// TIA Portal project "TiaProject-SortColors" (V17)

(* hardware
DEVICE "S7-1200 station_1"  S7-1200 Station
   slot 0: "Rack_0"  S7-1200 Rack  Rack  V1.0
   slot 1: "Brain"  CPU 1212C AC/DC/Rly  6ES7 212-1BE40-0XB0  V4.5
*)

// ===== PLC "Brain"  CPU 1212C AC/DC/Rly =====

VAR_GLOBAL   // PLC tag table "Steps"
   "X0" AT %M1.0 : Bool;
   "X1" AT %M1.1 : Bool;
   "X2" AT %M1.2 : Bool;
   "X3" AT %M1.3 : Bool;
   "X4" AT %M1.4 : Bool;
   "X5" AT %M1.5 : Bool;
   "X6" AT %M1.6 : Bool;
   "X7" AT %M1.7 : Bool;
   "X8" AT %M6.0 : Bool;
   "X9" AT %M6.1 : Bool;
   "X10" AT %M6.2 : Bool;
   "X11" AT %M6.3 : Bool;
   "X12" AT %M6.4 : Bool;
END_VAR

VAR_GLOBAL   // PLC tag table "I/O"
   "i1" AT %I0.0 : Bool;   // Belt Counter
   "i2" AT %I0.1 : Bool;   // Chromatic Entry
   "i3" AT %I0.3 : Bool;   // Chromatic Exit
   "i4" AT %IW64 : Int;   // Chromatic Sensor
   "i5" AT %I0.2 : Bool;   // White Presence
   "i6" AT %I0.6 : Bool;   // Red Presence
   "i7" AT %I0.7 : Bool;   // Blue Presence
   "start" AT %I0.5 : Bool;   // Start Button
   "stop" AT %I0.4 : Bool;   // Stop Button
   "Q1" AT %Q0.0 : Bool;   // Belt Motor
   "Q2" AT %Q0.1 : Bool;   // Compressor
   "Q3" AT %Q0.2 : Bool;   // White Jack
   "Q4" AT %Q0.4 : Bool;   // Red Jack
   "Q5" AT %Q0.5 : Bool;   // Blue Jack
END_VAR

VAR_GLOBAL   // PLC tag table "MemoryVariables"
   "BeltCounter" AT %MW2 : Int;   // Count the avancement of the belt.
   "LastChromaticValue" AT %MW4 : Int;   // Store the last value read by the chromatic sensor.
END_VAR

// folder: System blocks/Program resources

DATA_BLOCK "BeltCounterDB"   // DB1
{ S7_Optimized_Access := 'TRUE' }
AUTHOR : Simatic
FAMILY : IEC
NAME : CNTR
VERSION : 1.0
// stored: InstanceOfName IEC_COUNTER
"IEC_COUNTER"
BEGIN
END_DATA_BLOCK

DATA_BLOCK "TimerX3"   // DB2
{ S7_Optimized_Access := 'TRUE' }
AUTHOR : Simatic
FAMILY : IEC
NAME : IEC_TMR
VERSION : 1.0
// stored: InstanceOfName IEC_TIMER
"IEC_TIMER"
BEGIN
END_DATA_BLOCK

DATA_BLOCK "TimerX12"   // DB3
{ S7_Optimized_Access := 'TRUE' }
AUTHOR : Simatic
FAMILY : IEC
NAME : IEC_TMR
VERSION : 1.0
// stored: InstanceOfName IEC_TIMER
"IEC_TIMER"
BEGIN
END_DATA_BLOCK

// folder: (top level)

FUNCTION "CounterManager" : Void   // FC1, LAD
{ S7_Optimized_Access := 'TRUE' }
VERSION : 0.1
BEGIN

REGION Network 1: BeltCounterNetwork
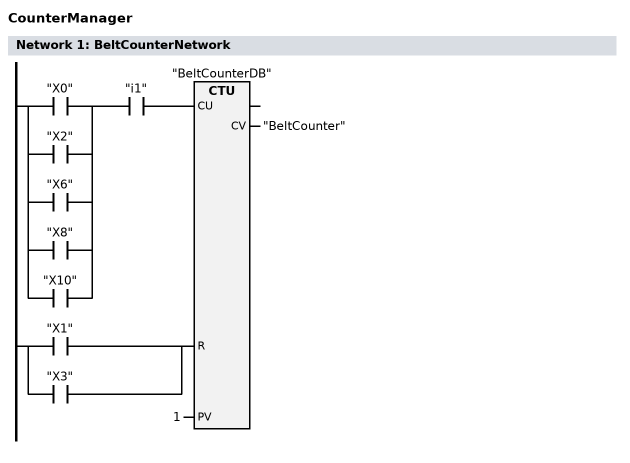
   "BeltCounterDB".CTU(CU := ("X0" OR "X2" OR "X6" OR "X8" OR "X10") AND "i1",
                       R := "X1" OR "X3",
                       PV := 1,
                       CV => "BeltCounter");
END_REGION
END_FUNCTION

FUNCTION "TimerManager" : Void   // FC2, LAD
{ S7_Optimized_Access := 'TRUE' }
VERSION : 0.1
BEGIN

REGION Network 1: TimerNetwork
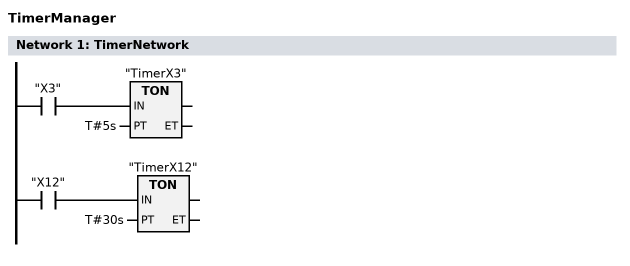
   "TimerX3".TON(IN := "X3", PT := T#5s);
   "TimerX12".TON(IN := "X12", PT := T#30s);
END_REGION
END_FUNCTION

FUNCTION "SetLastChromaticValue" : Void   // FC3, SCL
{ S7_Optimized_Access := 'TRUE' }
VERSION : 0.1
BEGIN
   "LastChromaticValue" := "i4";
END_FUNCTION

FUNCTION "OrderManager" : Void   // FC4, LAD
{ S7_Optimized_Access := 'TRUE' }
VERSION : 0.1
BEGIN

REGION Network 1: X0
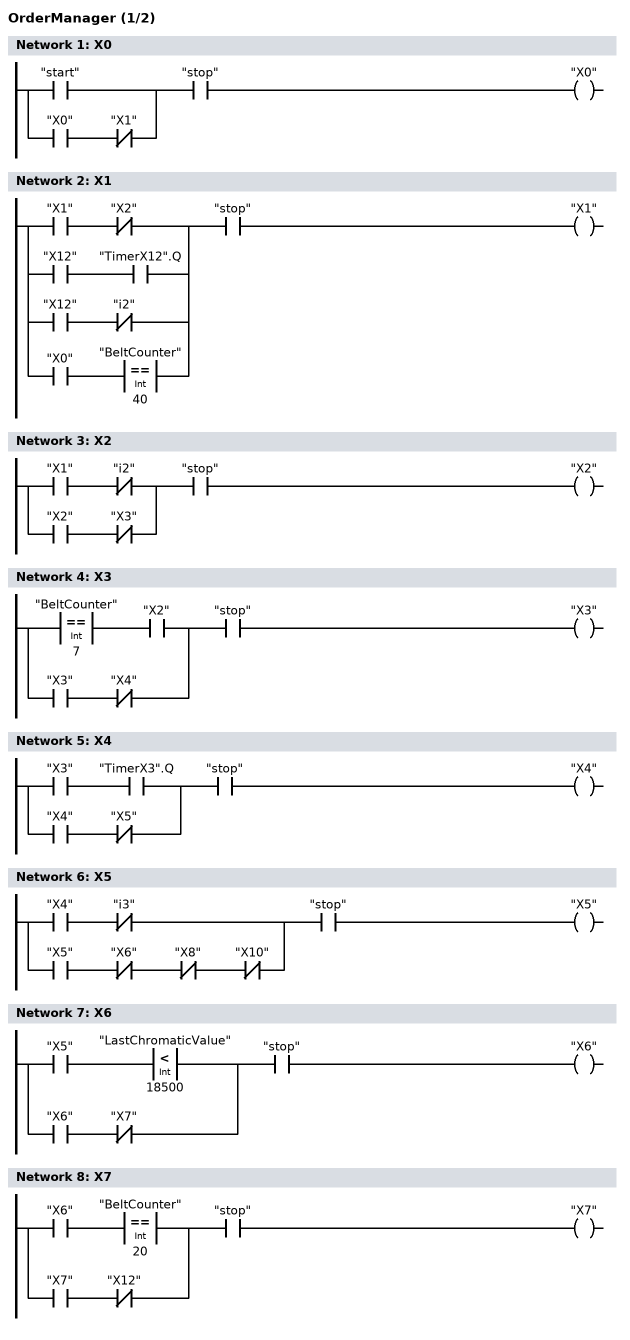
   RUNG wire#powerrail
      Contact( "start" )
      wire#w1
      Contact( "stop" )
      Coil( "X0" )
   END_RUNG
   RUNG wire#powerrail
      Contact( "X0" )
      I_Contact( "X1" )
   END_RUNG wire#w1
   // the same network as SCL:
   "X0" := ("start" OR ("X0" AND NOT "X1")) AND "stop";
END_REGION

REGION Network 2: X1
   RUNG wire#powerrail
      Contact( "X1" )
      I_Contact( "X2" )
      wire#w1
      Contact( "stop" )
      Coil( "X1" )
   END_RUNG
   RUNG wire#powerrail
      Contact( "X12" )
      Contact( "TimerX12".Q )
   END_RUNG wire#w1
   RUNG wire#powerrail
      Contact( "X12" )
      I_Contact( "i2" )
   END_RUNG wire#w1
   RUNG wire#powerrail
      Contact( "X0" )
      { S7_Templates := "SrcType := Int" } EQ_Contact(in1 := "BeltCounter", in2 := 40)
   END_RUNG wire#w1
   // the same network as SCL:
   "X1" := (("X1" AND NOT "X2") OR ("X12" AND "TimerX12".Q) OR ("X12" AND NOT "i2") OR ("X0" AND ("BeltCounter" = 40))) AND "stop";
END_REGION

REGION Network 3: X2
   RUNG wire#powerrail
      Contact( "X1" )
      I_Contact( "i2" )
      wire#w1
      Contact( "stop" )
      Coil( "X2" )
   END_RUNG
   RUNG wire#powerrail
      Contact( "X2" )
      I_Contact( "X3" )
   END_RUNG wire#w1
   // the same network as SCL:
   "X2" := (("X1" AND NOT "i2") OR ("X2" AND NOT "X3")) AND "stop";
END_REGION

REGION Network 4: X3
   RUNG wire#powerrail
      { S7_Templates := "SrcType := Int" } EQ_Contact(in1 := "BeltCounter", in2 := 7)
      Contact( "X2" )
      wire#w1
      Contact( "stop" )
      Coil( "X3" )
   END_RUNG
   RUNG wire#powerrail
      Contact( "X3" )
      I_Contact( "X4" )
   END_RUNG wire#w1
   // the same network as SCL:
   "X3" := ((("BeltCounter" = 7) AND "X2") OR ("X3" AND NOT "X4")) AND "stop";
END_REGION

REGION Network 5: X4
   RUNG wire#powerrail
      Contact( "X3" )
      Contact( "TimerX3".Q )
      wire#w1
      Contact( "stop" )
      Coil( "X4" )
   END_RUNG
   RUNG wire#powerrail
      Contact( "X4" )
      I_Contact( "X5" )
   END_RUNG wire#w1
   // the same network as SCL:
   "X4" := (("X3" AND "TimerX3".Q) OR ("X4" AND NOT "X5")) AND "stop";
END_REGION

REGION Network 6: X5
   RUNG wire#powerrail
      Contact( "X4" )
      I_Contact( "i3" )
      wire#w1
      Contact( "stop" )
      Coil( "X5" )
   END_RUNG
   RUNG wire#powerrail
      Contact( "X5" )
      I_Contact( "X6" )
      I_Contact( "X8" )
      I_Contact( "X10" )
   END_RUNG wire#w1
   // the same network as SCL:
   "X5" := (("X4" AND NOT "i3") OR ("X5" AND NOT "X6" AND NOT "X8" AND NOT "X10")) AND "stop";
END_REGION

REGION Network 7: X6
   RUNG wire#powerrail
      Contact( "X5" )
      { S7_Templates := "SrcType := Int" } LT_Contact(in1 := "LastChromaticValue", in2 := 18500)
      wire#w1
      Contact( "stop" )
      Coil( "X6" )
   END_RUNG
   RUNG wire#powerrail
      Contact( "X6" )
      I_Contact( "X7" )
   END_RUNG wire#w1
   // the same network as SCL:
   "X6" := (("X5" AND ("LastChromaticValue" < 18500)) OR ("X6" AND NOT "X7")) AND "stop";
END_REGION

REGION Network 8: X7
   RUNG wire#powerrail
      Contact( "X6" )
      { S7_Templates := "SrcType := Int" } EQ_Contact(in1 := "BeltCounter", in2 := 20)
      wire#w1
      Contact( "stop" )
      Coil( "X7" )
   END_RUNG
   RUNG wire#powerrail
      Contact( "X7" )
      I_Contact( "X12" )
   END_RUNG wire#w1
   // the same network as SCL:
   "X7" := (("X6" AND ("BeltCounter" = 20)) OR ("X7" AND NOT "X12")) AND "stop";
END_REGION

REGION Network 9: X8
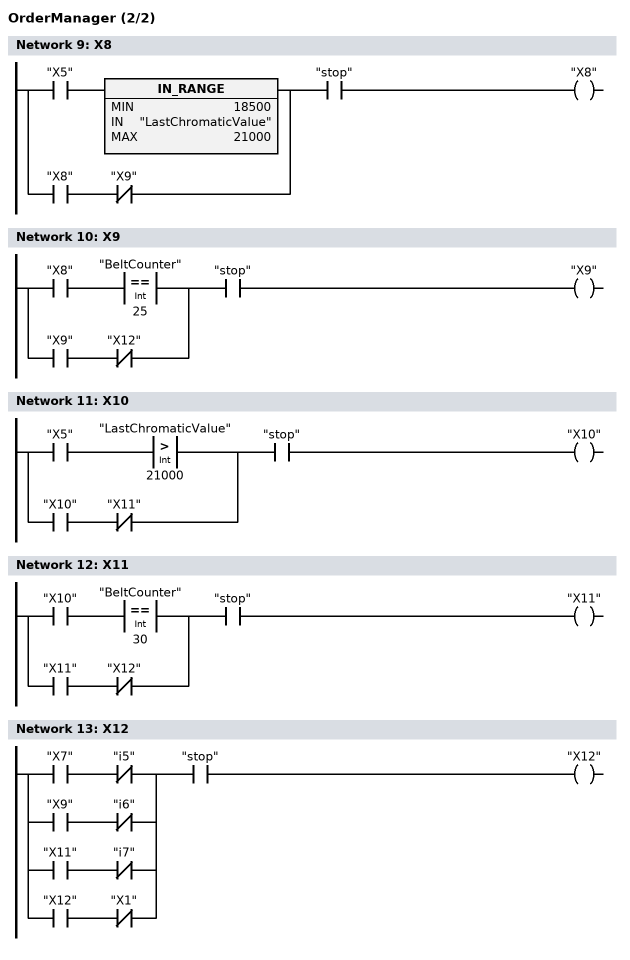
   RUNG wire#powerrail
      Contact( "X5" )
      { S7_Templates := "SrcType := Int" } InRange(min := 18500, in := "LastChromaticValue", max := 21000)
      wire#w1
      Contact( "stop" )
      Coil( "X8" )
   END_RUNG
   RUNG wire#powerrail
      Contact( "X8" )
      I_Contact( "X9" )
   END_RUNG wire#w1
   // the same network as SCL:
   "X8" := (("X5" AND (18500 <= "LastChromaticValue") AND ("LastChromaticValue" <= 21000)) OR ("X8" AND NOT "X9")) AND "stop";
END_REGION

REGION Network 10: X9
   RUNG wire#powerrail
      Contact( "X8" )
      { S7_Templates := "SrcType := Int" } EQ_Contact(in1 := "BeltCounter", in2 := 25)
      wire#w1
      Contact( "stop" )
      Coil( "X9" )
   END_RUNG
   RUNG wire#powerrail
      Contact( "X9" )
      I_Contact( "X12" )
   END_RUNG wire#w1
   // the same network as SCL:
   "X9" := (("X8" AND ("BeltCounter" = 25)) OR ("X9" AND NOT "X12")) AND "stop";
END_REGION

REGION Network 11: X10
   RUNG wire#powerrail
      Contact( "X5" )
      { S7_Templates := "SrcType := Int" } GT_Contact(in1 := "LastChromaticValue", in2 := 21000)
      wire#w1
      Contact( "stop" )
      Coil( "X10" )
   END_RUNG
   RUNG wire#powerrail
      Contact( "X10" )
      I_Contact( "X11" )
   END_RUNG wire#w1
   // the same network as SCL:
   "X10" := (("X5" AND ("LastChromaticValue" > 21000)) OR ("X10" AND NOT "X11")) AND "stop";
END_REGION

REGION Network 12: X11
   RUNG wire#powerrail
      Contact( "X10" )
      { S7_Templates := "SrcType := Int" } EQ_Contact(in1 := "BeltCounter", in2 := 30)
      wire#w1
      Contact( "stop" )
      Coil( "X11" )
   END_RUNG
   RUNG wire#powerrail
      Contact( "X11" )
      I_Contact( "X12" )
   END_RUNG wire#w1
   // the same network as SCL:
   "X11" := (("X10" AND ("BeltCounter" = 30)) OR ("X11" AND NOT "X12")) AND "stop";
END_REGION

REGION Network 13: X12
   RUNG wire#powerrail
      Contact( "X7" )
      I_Contact( "i5" )
      wire#w1
      Contact( "stop" )
      Coil( "X12" )
   END_RUNG
   RUNG wire#powerrail
      Contact( "X9" )
      I_Contact( "i6" )
   END_RUNG wire#w1
   RUNG wire#powerrail
      Contact( "X11" )
      I_Contact( "i7" )
   END_RUNG wire#w1
   RUNG wire#powerrail
      Contact( "X12" )
      I_Contact( "X1" )
   END_RUNG wire#w1
   // the same network as SCL:
   "X12" := (("X7" AND NOT "i5") OR ("X9" AND NOT "i6") OR ("X11" AND NOT "i7") OR ("X12" AND NOT "X1")) AND "stop";
END_REGION
END_FUNCTION

FUNCTION "SFCManager" : Void   // FC5, LAD
{ S7_Optimized_Access := 'TRUE' }
VERSION : 0.1
BEGIN

REGION Network 1: Activate Belt
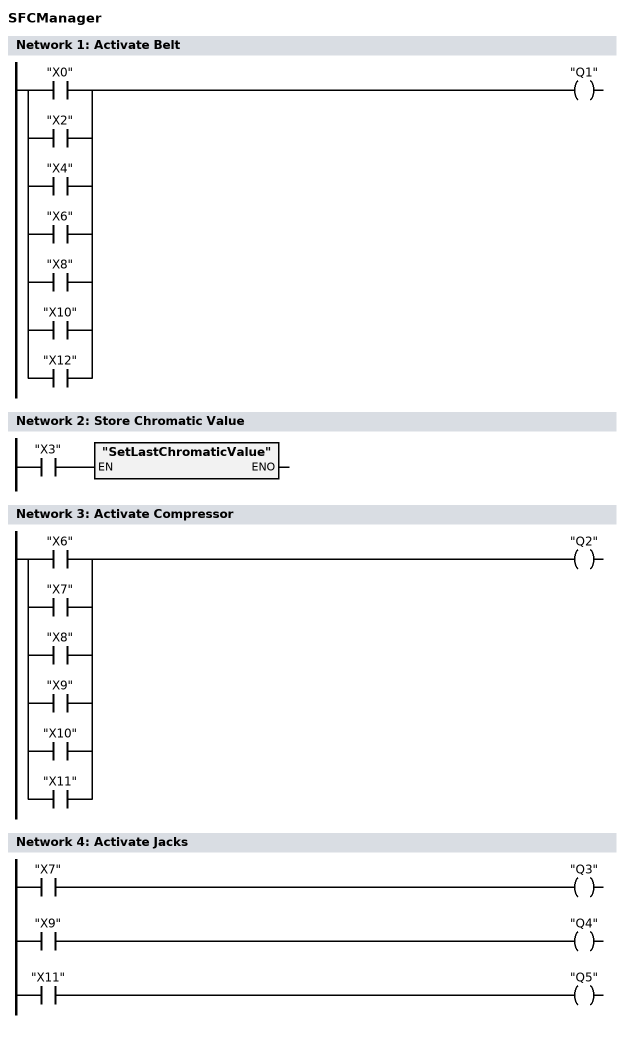
   RUNG wire#powerrail
      Contact( "X0" )
      wire#w1
      Coil( "Q1" )
   END_RUNG
   RUNG wire#powerrail
      Contact( "X2" )
   END_RUNG wire#w1
   RUNG wire#powerrail
      Contact( "X4" )
   END_RUNG wire#w1
   RUNG wire#powerrail
      Contact( "X6" )
   END_RUNG wire#w1
   RUNG wire#powerrail
      Contact( "X8" )
   END_RUNG wire#w1
   RUNG wire#powerrail
      Contact( "X10" )
   END_RUNG wire#w1
   RUNG wire#powerrail
      Contact( "X12" )
   END_RUNG wire#w1
   // the same network as SCL:
   "Q1" := "X0" OR "X2" OR "X4" OR "X6" OR "X8" OR "X10" OR "X12";
END_REGION

REGION Network 2: Store Chromatic Value
   RUNG wire#powerrail
      Contact( "X3" )
      "SetLastChromaticValue"()
   END_RUNG
   // the same network as SCL:
   IF "X3" THEN "SetLastChromaticValue"(); END_IF;
END_REGION

REGION Network 3: Activate Compressor
   RUNG wire#powerrail
      Contact( "X6" )
      wire#w1
      Coil( "Q2" )
   END_RUNG
   RUNG wire#powerrail
      Contact( "X7" )
   END_RUNG wire#w1
   RUNG wire#powerrail
      Contact( "X8" )
   END_RUNG wire#w1
   RUNG wire#powerrail
      Contact( "X9" )
   END_RUNG wire#w1
   RUNG wire#powerrail
      Contact( "X10" )
   END_RUNG wire#w1
   RUNG wire#powerrail
      Contact( "X11" )
   END_RUNG wire#w1
   // the same network as SCL:
   "Q2" := "X6" OR "X7" OR "X8" OR "X9" OR "X10" OR "X11";
END_REGION

REGION Network 4: Activate Jacks
   RUNG wire#powerrail
      Contact( "X7" )
      Coil( "Q3" )
   END_RUNG
   RUNG wire#powerrail
      Contact( "X9" )
      Coil( "Q4" )
   END_RUNG
   RUNG wire#powerrail
      Contact( "X11" )
      Coil( "Q5" )
   END_RUNG
   // the same network as SCL:
   "Q3" := "X7";
   "Q4" := "X9";
   "Q5" := "X11";
END_REGION
END_FUNCTION

ORGANIZATION_BLOCK "Main"   // OB1, LAD, ProgramCycle
TITLE = "Main Program Sweep (Cycle)"
{ S7_Optimized_Access := 'TRUE' }
VERSION : 0.1
   VAR_INPUT
      Initial_Call : Bool;   // Initial call of this OB
      Remanence : Bool;   // =True, if remanent data are available
   END_VAR
   VAR_TEMP   // added for the SCL form of the ladder/FBD networks
      _w1 : Bool;
      _w2 : Bool;
      _w3 : Bool;
   END_VAR
BEGIN

REGION Network 1
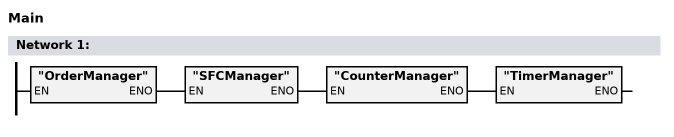
   RUNG wire#powerrail
      "OrderManager"()
      "SFCManager"()
      "CounterManager"()
      "TimerManager"()
   END_RUNG
   // the same network as SCL:
   "OrderManager"(ENO => #_w1);
   "SFCManager"(EN := #_w1, ENO => #_w2);
   "CounterManager"(EN := #_w2, ENO => #_w3);
   IF #_w3 THEN "TimerManager"(); END_IF;
END_REGION
END_ORGANIZATION_BLOCK